Staubli VAL3: italiano.dtx

public string No = "No"
public string Yes = "Si"
public mdesc nom_speed = {rmax=9999, blend=off}
